// TIA Portal V17 export
// export: Created 2024-08-07T21:44:11.3165906Z, ExportSetting WithDefaults, DisplayName Totally Integrated Automation Portal, DisplayVersion V17 Update 7, DisplayName TIA Portal Openness, DisplayVersion V17 Update 7, DisplayName TIA Portal Version Control Interface, DisplayVersion V17, DisplayName SINAMICS Startdrive Advanced, DisplayVersion V17 SP2, DisplayName SINAMICS Startdrive G110M, G120, G120C, G120D, G120P, G115D, DisplayVersion V17 SP2, DisplayName SINAMICS Startdrive G130, G150, S120, S150, SINAMICS MV, S210, DisplayVersion V17 SP2, DisplayName STEP 7 Professional, DisplayVersion V17 Update 7, DisplayName STEP 7 Safety, DisplayVersion V17 Update 6, DisplayName WinCC Advanced / Unified PC, DisplayVersion V17 Update 7
DATA_BLOCK "1. DMC_setConnection_DB"   // DB2002
VERSION : 0.1
// stored: AutoNumber false, DBAccessibleFromOPCUA true, DBAccessibleFromWebserver true, InstanceOfName 1. DMC_setConnection, InstanceOfType FB
"1. DMC_setConnection"
   // VAR
   //    Connection : Struct
   //       IPAddress : WString;
   //       ServerPort : WString;
   //       PlantID : WString;
   //       PLC_ID : WString;
   //       OperationMode : Bool;
   //    END_STRUCT;
   //    Controllers : Struct
   //       opcUaConnect : Bool;
   //       opcUaMethodCall : Bool;
   //       opcUaMethodIndex : SInt;
   //       opcUaConnected { S7_SetPoint := 'True'} : Bool;
   //       opcUaDone : Bool;
   //       opcUaBusy : Bool;
   //       opcUaError : Bool;
   //       opcUaStatus : Word;
   //       opcUaDiagnostics : "typeFbDiagnostics";
   //    END_STRUCT;
   //    Auxiliar : Struct
   //       endpointTemp : String[254];
   //       idx : Int;
   //       timeout : Bool;
   //       reconnectionTimeout : Bool;
   //       tryAgain : Bool;
   //    END_STRUCT;
   //    Timers : Struct
   //       timeoutCallMethod : TON_TIME;
   //       forceReconnection { S7_SetPoint := 'True'} : TON_TIME;
   //       tryAgain { S7_SetPoint := 'True'} : TON_TIME;
   //    END_STRUCT;
   //    CallBuffer : Array[0..9] of Bool;
   // END_VAR
BEGIN
END_DATA_BLOCK
